// TIA Portal project "lab3" (V17)

(* hardware
DEVICE "S7-1500/ET200MP station_1"  S7-1500 station
   slot 0: "Rail_0"  Rack  6ES7 590-1***0-0AA0
   slot 1: "PLC_1"  CPU 1518-4 PN/DP  6ES7 518-4AP00-0AB0  V2.9
      slot 3: "CPU display_1"  6ES7591-1BA00-0AA0
      slot 32768: "PROFINET interface_1"  X1
         slot 32769: "Port_1"  X1 P1
         slot 32770: "Port_2"  X1 P2
      slot 33024: "PROFINET interface_2"  X2
         slot 33025: "Port_1"  X2 P1
      slot 33280: "PROFINET interface GBIT_3"  X3
         slot 33281: "Port_1"  X3 P1
      slot 33536: "DP interface_1"  X4
      slot 34817: "Virtual CP interface port_1"  Virtual CP interface port  Virtual CP interface port
*)

// ===== PLC "PLC_1"  CPU 1518-4 PN/DP =====

VAR_GLOBAL   // PLC tag table "Default tag table"
   "Tag_1" AT %I0.0 : Bool;
   "Tag_2" AT %Q0.3 : Bool;
   "Tag_3" AT %M50.0 : Bool;
   "Tag_4" AT %M50.1 : Bool;
   "Tag_5" AT %M50.2 : Bool;
   "Tag_6" AT %Q0.4 : Bool;
   "Tag_7" AT %I1.0 : Bool;
   "Tag_8" AT %M51.0 : Bool;
   "Tag_9" AT %M51.1 : Bool;
   "Tag_10" AT %M52.0 : Bool;
   "Tag_11" AT %M52.1 : Bool;
   "Tag_12" AT %Q0.0 : Bool;
   "Tag_13" AT %M52.2 : Bool;
   "Tag_14" AT %M52.3 : Bool;
END_VAR

DATA_BLOCK "TON_miganie_FB_DB"   // DB9
{ S7_Optimized_Access := 'TRUE' }
VERSION : 0.1
// stored: InstanceOfName TON_miganie_FB
"TON_miganie_FB"
BEGIN
END_DATA_BLOCK

// folder: System blocks/Program resources

DATA_BLOCK "IEC_Timer_0_DB"   // DB1
{ S7_Optimized_Access := 'TRUE' }
AUTHOR : Simatic
FAMILY : IEC
NAME : IEC_TMR
VERSION : 1.0
// stored: InstanceOfName IEC_TIMER
"IEC_TIMER"
BEGIN
END_DATA_BLOCK

DATA_BLOCK "IEC_Timer_0_DB_1"   // DB2
{ S7_Optimized_Access := 'TRUE' }
AUTHOR : Simatic
FAMILY : IEC
NAME : IEC_TMR
VERSION : 1.0
// stored: InstanceOfName IEC_TIMER
"IEC_TIMER"
BEGIN
END_DATA_BLOCK

DATA_BLOCK "IEC_Timer_0_DB_2"   // DB3
{ S7_Optimized_Access := 'TRUE' }
AUTHOR : Simatic
FAMILY : IEC
NAME : IEC_TMR
VERSION : 1.0
// stored: InstanceOfName IEC_TIMER
"IEC_TIMER"
BEGIN
END_DATA_BLOCK

DATA_BLOCK "IEC_Timer_0_DB_3"   // DB4
{ S7_Optimized_Access := 'TRUE' }
AUTHOR : Simatic
FAMILY : IEC
NAME : IEC_TMR
VERSION : 1.0
// stored: InstanceOfName IEC_TIMER
"IEC_TIMER"
BEGIN
END_DATA_BLOCK

DATA_BLOCK "IEC_Timer_0_DB_4"   // DB5
{ S7_Optimized_Access := 'TRUE' }
AUTHOR : Simatic
FAMILY : IEC
NAME : IEC_TMR
VERSION : 1.0
// stored: InstanceOfName IEC_TIMER
"IEC_TIMER"
BEGIN
END_DATA_BLOCK

DATA_BLOCK "IEC_Timer_0_DB_5"   // DB6
{ S7_Optimized_Access := 'TRUE' }
AUTHOR : Simatic
FAMILY : IEC
NAME : IEC_TMR
VERSION : 1.0
// stored: InstanceOfName IEC_TIMER
"IEC_TIMER"
BEGIN
END_DATA_BLOCK

DATA_BLOCK "IEC_Timer_0_DB_6"   // DB7
{ S7_Optimized_Access := 'TRUE' }
AUTHOR : Simatic
FAMILY : IEC
NAME : IEC_TMR
VERSION : 1.0
// stored: InstanceOfName IEC_TIMER
"IEC_TIMER"
BEGIN
END_DATA_BLOCK

DATA_BLOCK "IEC_Timer_0_DB_7"   // DB8
{ S7_Optimized_Access := 'TRUE' }
AUTHOR : Simatic
FAMILY : IEC
NAME : IEC_TMR
VERSION : 1.0
// stored: InstanceOfName IEC_TIMER
"IEC_TIMER"
BEGIN
END_DATA_BLOCK

// folder: (top level)

FUNCTION_BLOCK "TON_miganie_FB"   // FB1, LAD
{ S7_Optimized_Access := 'TRUE' }
VERSION : 0.1
   VAR_INPUT
      Okres : DInt;
      IN : Bool;
      "Wypelnienie [%]" : Int;
   END_VAR
   VAR_OUTPUT
      Output : Bool;
   END_VAR
   VAR
      temp : Bool;
      temp2 : Bool;
   END_VAR
   VAR_TEMP
      TON_Out : Bool;
      Wypelnienie_DInt : DInt;
      Wypelnienie_Temp : DInt;
   END_VAR
   VAR_TEMP   // added for the SCL form of the ladder/FBD networks
      _w1 : Bool;
      _w2 : Bool;
   END_VAR
BEGIN

REGION Network 1
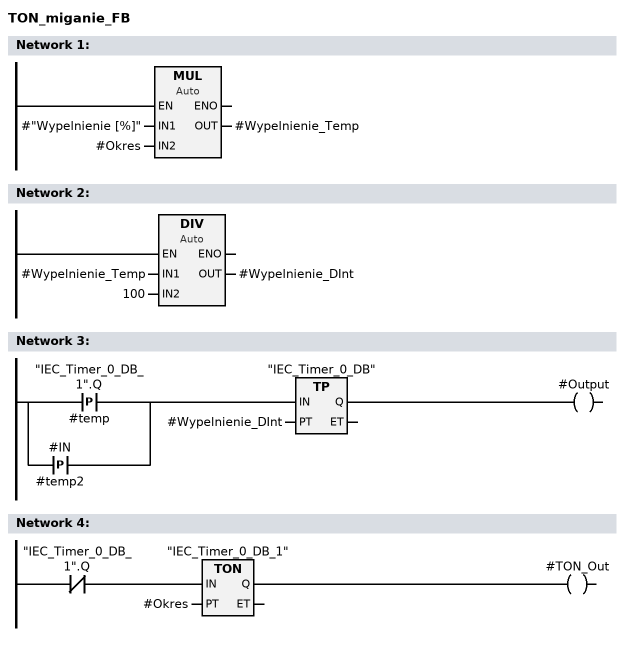
   RUNG wire#powerrail
      Mul(in1 := #"Wypelnienie [%]", in2 := #Okres, out => #Wypelnienie_Temp)
   END_RUNG
   // the same network as SCL:
   #Wypelnienie_Temp := #"Wypelnienie [%]" * #Okres;
END_REGION

REGION Network 2
   RUNG wire#powerrail
      Div(in1 := #Wypelnienie_Temp, in2 := 100, out => #Wypelnienie_DInt)
   END_RUNG
   // the same network as SCL:
   #Wypelnienie_DInt := #Wypelnienie_Temp / 100;
END_REGION

REGION Network 3
   #_w1 := "IEC_Timer_0_DB_1".Q AND NOT #temp;   // rising edge of "IEC_Timer_0_DB_1".Q
   #temp := "IEC_Timer_0_DB_1".Q;
   #_w2 := #IN AND NOT #temp2;   // rising edge of #IN
   #temp2 := #IN;
   "IEC_Timer_0_DB".TP(IN := #_w1 OR #_w2, PT := #Wypelnienie_DInt);
   #Output := "IEC_Timer_0_DB".Q;
END_REGION

REGION Network 4
   "IEC_Timer_0_DB_1".TON(IN := NOT "IEC_Timer_0_DB_1".Q, PT := #Okres);
   #TON_Out := "IEC_Timer_0_DB_1".Q;
END_REGION
END_FUNCTION_BLOCK

FUNCTION "TON_miganie" : Void   // FC1, LAD
{ S7_Optimized_Access := 'TRUE' }
VERSION : 0.1
   VAR_INPUT
      Okres : DInt;
      IN : Bool;
      "Wypelnienie [%]" : Int;
   END_VAR
   VAR_OUTPUT
      Output : Bool;
   END_VAR
   VAR_TEMP
      TON_Out : Bool;
      Wypelnienie_DInt : DInt;
      Wypelnienie_Temp : DInt;
      temp : Bool;
      temp2 : Bool;
   END_VAR
   VAR_TEMP   // added for the SCL form of the ladder/FBD networks
      _w1 : Bool;
      _w2 : Bool;
   END_VAR
BEGIN

REGION Network 1
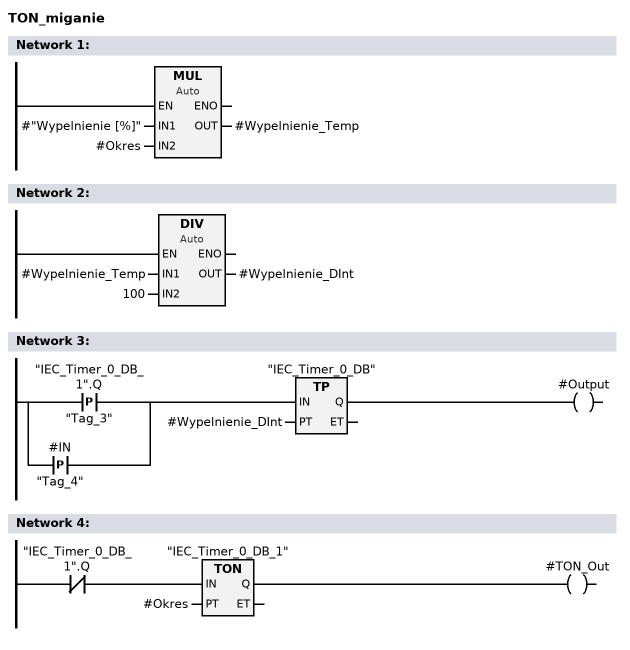
   RUNG wire#powerrail
      Mul(in1 := #"Wypelnienie [%]", in2 := #Okres, out => #Wypelnienie_Temp)
   END_RUNG
   // the same network as SCL:
   #Wypelnienie_Temp := #"Wypelnienie [%]" * #Okres;
END_REGION

REGION Network 2
   RUNG wire#powerrail
      Div(in1 := #Wypelnienie_Temp, in2 := 100, out => #Wypelnienie_DInt)
   END_RUNG
   // the same network as SCL:
   #Wypelnienie_DInt := #Wypelnienie_Temp / 100;
END_REGION

REGION Network 3
   #_w1 := "IEC_Timer_0_DB_1".Q AND NOT "Tag_3";   // rising edge of "IEC_Timer_0_DB_1".Q
   "Tag_3" := "IEC_Timer_0_DB_1".Q;
   #_w2 := #IN AND NOT "Tag_4";   // rising edge of #IN
   "Tag_4" := #IN;
   "IEC_Timer_0_DB".TP(IN := #_w1 OR #_w2, PT := #Wypelnienie_DInt);
   #Output := "IEC_Timer_0_DB".Q;
END_REGION

REGION Network 4
   "IEC_Timer_0_DB_1".TON(IN := NOT "IEC_Timer_0_DB_1".Q, PT := #Okres);
   #TON_Out := "IEC_Timer_0_DB_1".Q;
END_REGION
END_FUNCTION

FUNCTION "TOF_miganie" : Void   // FC2, LAD
{ S7_Optimized_Access := 'TRUE' }
VERSION : 0.1
   VAR_INPUT
      Wlacz : Bool;
      Wypelnienie : Time;
      Okres : Time;
   END_VAR
   VAR_OUTPUT
      Output : Bool;
   END_VAR
   VAR_TEMP
      TOF_Out : Bool;
   END_VAR
   VAR_TEMP   // added for the SCL form of the ladder/FBD networks
      _w1 : Bool;
      _w2 : Bool;
   END_VAR
BEGIN

REGION Network 1
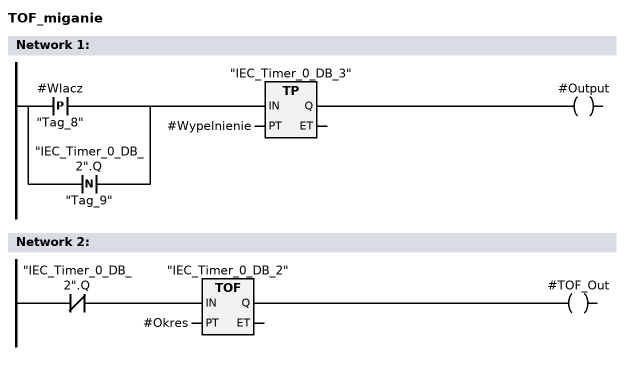
   #_w1 := #Wlacz AND NOT "Tag_8";   // rising edge of #Wlacz
   "Tag_8" := #Wlacz;
   #_w2 := NOT "IEC_Timer_0_DB_2".Q AND "Tag_9";   // falling edge of "IEC_Timer_0_DB_2".Q
   "Tag_9" := "IEC_Timer_0_DB_2".Q;
   "IEC_Timer_0_DB_3".TP(IN := #_w1 OR #_w2, PT := #Wypelnienie);
   #Output := "IEC_Timer_0_DB_3".Q;
END_REGION

REGION Network 2
   "IEC_Timer_0_DB_2".TOF(IN := NOT "IEC_Timer_0_DB_2".Q, PT := #Okres);
   #TOF_Out := "IEC_Timer_0_DB_2".Q;
END_REGION
END_FUNCTION

FUNCTION "klatka_schodowa" : Void   // FC3, LAD
{ S7_Optimized_Access := 'TRUE' }
VERSION : 0.1
   VAR_INPUT
      Przycisk : Bool;
   END_VAR
   VAR_OUTPUT
      Out : Bool;
   END_VAR
   VAR_TEMP
      Out1 : Bool;
      Out2 : Bool;
      temp : Bool;
   END_VAR
   VAR_TEMP   // added for the SCL form of the ladder/FBD networks
      _w1 : Bool;
   END_VAR
BEGIN

REGION Network 1
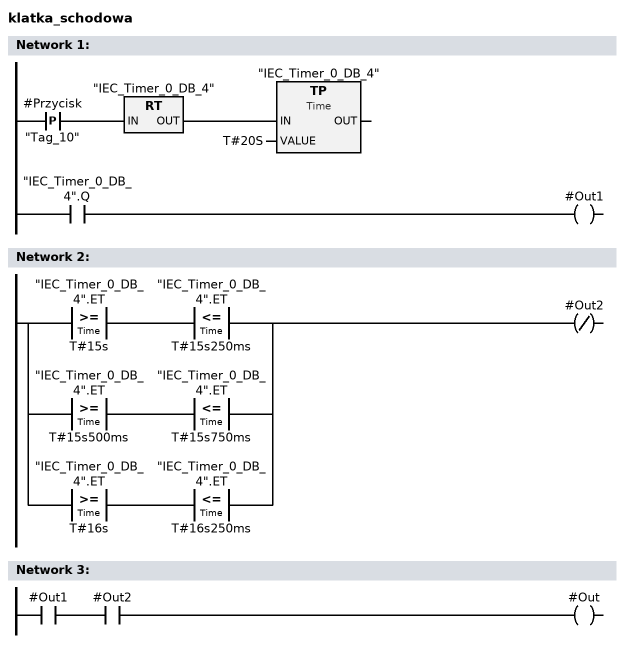
   #_w1 := #Przycisk AND NOT "Tag_10";   // rising edge of #Przycisk
   "Tag_10" := #Przycisk;
   IF #_w1 THEN RESET_TIMER("IEC_Timer_0_DB_4"); END_IF;
   "IEC_Timer_0_DB_4".TP(IN := #_w1, PT := T#20S);   // TP coil
   #Out1 := "IEC_Timer_0_DB_4".Q;
END_REGION

REGION Network 2
   RUNG wire#powerrail
      { S7_Templates := "SrcType := Time" } GE_Contact(in1 := "IEC_Timer_0_DB_4".ET, in2 := T#15s)
      { S7_Templates := "SrcType := Time" } LE_Contact(in1 := "IEC_Timer_0_DB_4".ET, in2 := T#15s250ms)
      wire#w1
      I_Coil( #Out2 )
   END_RUNG
   RUNG wire#powerrail
      { S7_Templates := "SrcType := Time" } GE_Contact(in1 := "IEC_Timer_0_DB_4".ET, in2 := T#15s500ms)
      { S7_Templates := "SrcType := Time" } LE_Contact(in1 := "IEC_Timer_0_DB_4".ET, in2 := T#15s750ms)
   END_RUNG wire#w1
   RUNG wire#powerrail
      { S7_Templates := "SrcType := Time" } GE_Contact(in1 := "IEC_Timer_0_DB_4".ET, in2 := T#16s)
      { S7_Templates := "SrcType := Time" } LE_Contact(in1 := "IEC_Timer_0_DB_4".ET, in2 := T#16s250ms)
   END_RUNG wire#w1
   // the same network as SCL:
   #Out2 := NOT ((("IEC_Timer_0_DB_4".ET >= T#15s) AND ("IEC_Timer_0_DB_4".ET <= T#15s250ms)) OR (("IEC_Timer_0_DB_4".ET >= T#15s500ms) AND ("IEC_Timer_0_DB_4".ET <= T#15s750ms)) OR (("IEC_Timer_0_DB_4".ET >= T#16s) AND ("IEC_Timer_0_DB_4".ET <= T#16s250ms)));
END_REGION

REGION Network 3
   RUNG wire#powerrail
      Contact( #Out1 )
      Contact( #Out2 )
      Coil( #Out )
   END_RUNG
   // the same network as SCL:
   #Out := #Out1 AND #Out2;
END_REGION
END_FUNCTION

FUNCTION "T_delay" : Void   // FC4, LAD
{ S7_Optimized_Access := 'TRUE' }
VERSION : 0.1
   VAR_INPUT
      IN : Bool;
      PT_ON : Time;
      PT_OFF : Time;
   END_VAR
   VAR_OUTPUT
      OUT : Bool;
   END_VAR
   VAR_TEMP
      TON_OUT : Bool;
   END_VAR
BEGIN

REGION Network 1
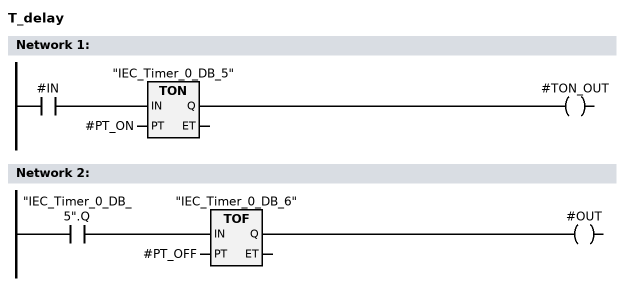
   "IEC_Timer_0_DB_5".TON(IN := #IN, PT := #PT_ON);
   #TON_OUT := "IEC_Timer_0_DB_5".Q;
END_REGION

REGION Network 2
   "IEC_Timer_0_DB_6".TOF(IN := "IEC_Timer_0_DB_5".Q, PT := #PT_OFF);
   #OUT := "IEC_Timer_0_DB_6".Q;
END_REGION
END_FUNCTION

FUNCTION "T_impuls" : Void   // FC5, LAD
{ S7_Optimized_Access := 'TRUE' }
VERSION : 0.1
   VAR_INPUT
      PT : DInt;
      IN : Bool;
   END_VAR
   VAR_OUTPUT
      Out : Bool;
   END_VAR
   VAR_TEMP
      temp : Bool;
   END_VAR
BEGIN

REGION Network 1
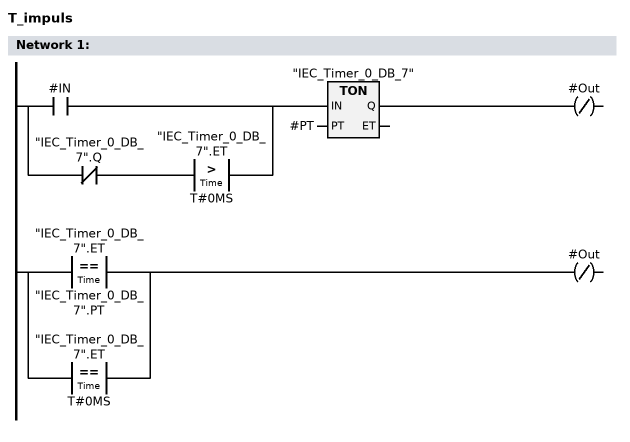
   "IEC_Timer_0_DB_7".TON(IN := #IN OR (NOT "IEC_Timer_0_DB_7".Q AND ("IEC_Timer_0_DB_7".ET > T#0MS)),
                          PT := #PT);
   #Out := NOT "IEC_Timer_0_DB_7".Q;
   #Out := NOT (("IEC_Timer_0_DB_7".ET = "IEC_Timer_0_DB_7".PT) OR ("IEC_Timer_0_DB_7".ET = T#0MS));
END_REGION
END_FUNCTION

ORGANIZATION_BLOCK "Main"   // OB1, LAD, ProgramCycle
TITLE = "Main Program Sweep (Cycle)"
{ S7_Optimized_Access := 'TRUE' }
VERSION : 0.1
   VAR_INPUT
      Initial_Call : Bool;   // Initial call of this OB
      Remanence : Bool;   // =True, if remanent data are available
   END_VAR
BEGIN

REGION Network 1
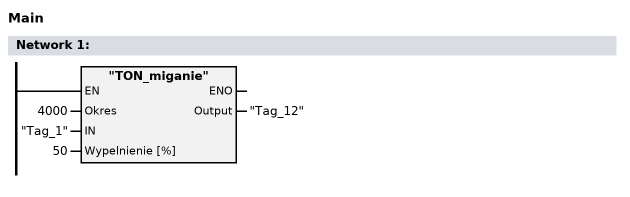
   RUNG wire#powerrail
      "TON_miganie"(Okres := 4000, IN := "Tag_1", "Wypelnienie [%]" := 50, Output => "Tag_12")
   END_RUNG
   // the same network as SCL:
   "TON_miganie"(Okres := 4000, IN := "Tag_1", "Wypelnienie [%]" := 50, Output => "Tag_12");
END_REGION
END_ORGANIZATION_BLOCK